(* Logix 5000 project; controller flash vendor 1 type 14 code 150 rev 30.11; software revision 30.00 *)

TASK MainTask (continuous, watchdog 500 ms) : MainProgram

MODULES
   Local : vendor 1 type 14 code 150 (Compact 0, rev 30.11)
      Discrete_IO : Embedded (Compact 1, rev 3.1, Output RPI 20 ms)
      Analog_IO : Embedded (Compact 2, rev 1.1, Output RPI 80 ms)
      Counters : Embedded (Compact 3, rev 1.1, Output RPI 20 ms)
END_MODULES

PROGRAM MainProgram   (* main routine MainRoutine *)
VAR
   ARRAY_1 : DINT[34] := ([1] := 1, [2] := 2, [3] := 4, [4] := 8, [5] := 16, [6] := 32, [7] := 64, [8] := 128, [9] := 256, [10] := 512, [11] := 1024, [12] := 2048, [13] := 4096, [14] := 8192, [15] := 16384, [16] := 32768, [17] := 16384, [18] := 8192, [19] := 4096, [20] := 2048, [21] := 1024, [22] := 512, [23] := 256, [24] := 128, [25] := 64, [26] := 32, [27] := 16, [28] := 8, [29] := 4, [30] := 2, [31] := 1);
   controll : CONTROL := (LEN := 31, POS := 13);
   output : DINT := 4096;
   T4_1 : TIMER := (PRE := 100, ACC := 97, EN := 1, TT := 1);   // ON TIME
   T4_2 : TIMER := (PRE := 100);   // TIME OFF
END_VAR

ROUTINE MainRoutine   (* ladder *)
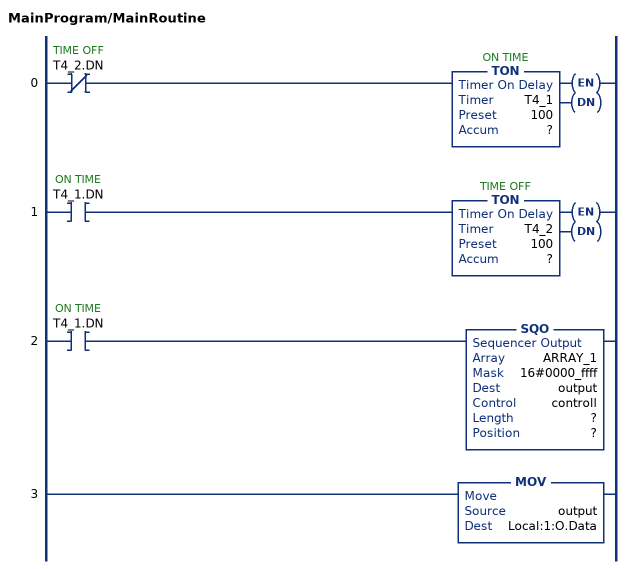
   0: XIO(T4_2.DN)TON(T4_1,?,?);
   1: XIC(T4_1.DN)TON(T4_2,?,?);
   2: XIC(T4_1.DN)SQO(ARRAY_1,16#0000_ffff,output,controll,?,?);
   3: MOV(output,Local:1:O.Data);
END_ROUTINE
END_PROGRAM
